# EPICS substitutions: AMI18001.substitutions
file AMI1800.template
{
pattern {S, TA, DN}
        {SECAGE, SE, AMI18001}
}
